// TIA Portal V20 export
// export: Created 2026-04-28T10:05:08.0016454Z, ExportSetting WithDefaults, DisplayName Totally Integrated Automation Portal, DisplayVersion V20, DisplayName TIA Portal Openness, DisplayVersion V20, DisplayName TIA Portal Version Control Interface, DisplayVersion V20, DisplayName SINAMICS Startdrive Advanced, DisplayVersion V20, DisplayName SINAMICS Startdrive G130, G150, S120, S150, SINAMICS MV, G220, S200, S210, DisplayVersion V20, DisplayName SINAMICS Startdrive G110M, G120, G120C, G120D, G120P, G115D, DisplayVersion V20, DisplayName STEP 7 Professional, DisplayVersion V20, DisplayName STEP 7 Safety, DisplayVersion V20, DisplayName WinCC Basic/Comfort/Advanced, DisplayVersion V20, DisplayName WinCC Unified, DisplayVersion V20
TYPE "Diag_EinAusVentile"
TITLE = EinAus-Ventile
// stored: IsFailsafeCompliant false
   STRUCT
      "Name" : String;   // Name/Bezeichner des Ventils
      EinAus : Bool;   // Ansteuerung von der SPS aktiv oder inaktiv
      Offen : Bool;   // Ventil geöffnet
      Geschlossen : Bool;   // Ventil geschlossen
      IntVisu : Int;   // 0: Ventil aus/nicht geschalten/Standardwert 1: Ventil aktiv 2: Fehler
      Fehler : Bool;   // Ventil Klemmt oder SPS Ausgang defekt.
   END_STRUCT;
END_TYPE
